{attribute 'qualified_only'}
VAR_GLOBAL
	
(*BUS COUPLER 8 OUTPUTS REFER TO SCHEMATIC CX8190-EL1859-1*)
EL1859_1			AT %Q*		:WORD;

(*BUS COUPLER 8 OUTPUTS REFER TO SCHEMATIC CX8190-EL1859-2*)
EL1859_2			AT %Q*		:WORD;

END_VAR

(* stored: Version 1.1.0.1, ProductVersion 3.1.4024.11
   GVL OUTPUT: Id {6ec63b1c-3068-4b6b-be81-5c9d025cb7fc} *)
